TYPE Outbound :
STRUCT
	roller	: Roller;
	photo_sensor	: FB_DigitalInput;
END_STRUCT
END_TYPE

(* stored: Version 1.1.0.1, ProductVersion 3.1.4024.12
   DUT Outbound: Id {358b3f71-70a1-4970-bff2-29ec36b29fb6} *)
